TYPE "MotorCtrl"
VERSION : 0.1
// Block: MotorCtrl
   STRUCT
      SafeStop : Bool;
      Rst : Bool;
      Run : Bool;
   END_STRUCT;

END_TYPE
